{attribute addProperty BoxType "EJ1957-0000-0017"}
{attribute addProperty Id "FSoE_InputsFSoE_Inputs_E4152F08567FSoE_OutputsFSoE_Outputs_865CD7FA567"}
{attribute addProperty CRC "3039541012"}
{attribute addProperty SizeInBites "112"}
{attribute addProperty SizeInBytes "14"}
TYPE Module_1_FSOE_B52BB714 :
STRUCT
	{attribute addProperty Name "FSoE_Inputs"}
	FSoE_Inputs  : FSoE_Inputs_E4152F08;
	{attribute addProperty Name "FSoE_Outputs"}
	FSoE_Outputs  : FSoE_Outputs_865CD7FA;
END_STRUCT
END_TYPE

(* stored: Version 1.2.0.0, ProductVersion 3.1.4024.9
   DUT Module_1_FSOE_B52BB714: Id {6cd79a23-a4fd-462e-b2e0-0ca6f044c210} *)
